% RSLogix 500 project horizontal_tank_integer.RSS, saved by version 8.30.00.16 %
PROJECT "UNTITLED"    % processor: Bul.1763 MicroLogix 1100 Series A %

PROGRAM FILES
  LAD 2   2 rungs
  LAD 255 "ONEDEPTH"  10 rungs

DATA FILES
  O0 OUTPUT  4 elements
  I1 INPUT  6 elements
  S2 STATUS  66 elements
  B3 BINARY  1 elements
  T4 TIMER  1 elements
  C5 COUNTER  1 elements
  R6 CONTROL  1 elements
  N7 INTEGER  20 elements
  F8 FLOAT  1 elements
  F254   128 elements
  N255   256 elements

LADDER 2
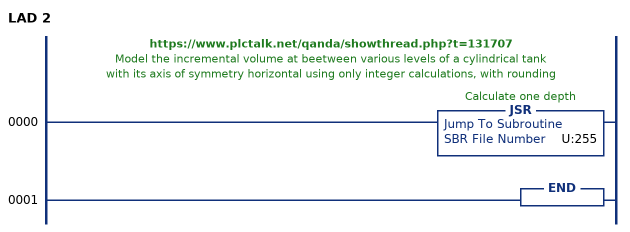
% Rung: 0 %
% TITLE: https://www.plctalk.net/qanda/showthread.php?t=131707 %
% Model the incremental volume at beetween various levels of a cylindrical tank
% with its axis of symmetry horizontal using only integer calculations, with rounding %
SOR JSR U:255 EOR
%   U:255  "Calculate one depth" %
% Rung: 1 %
SOR END EOR

LADDER 255 "ONEDEPTH"
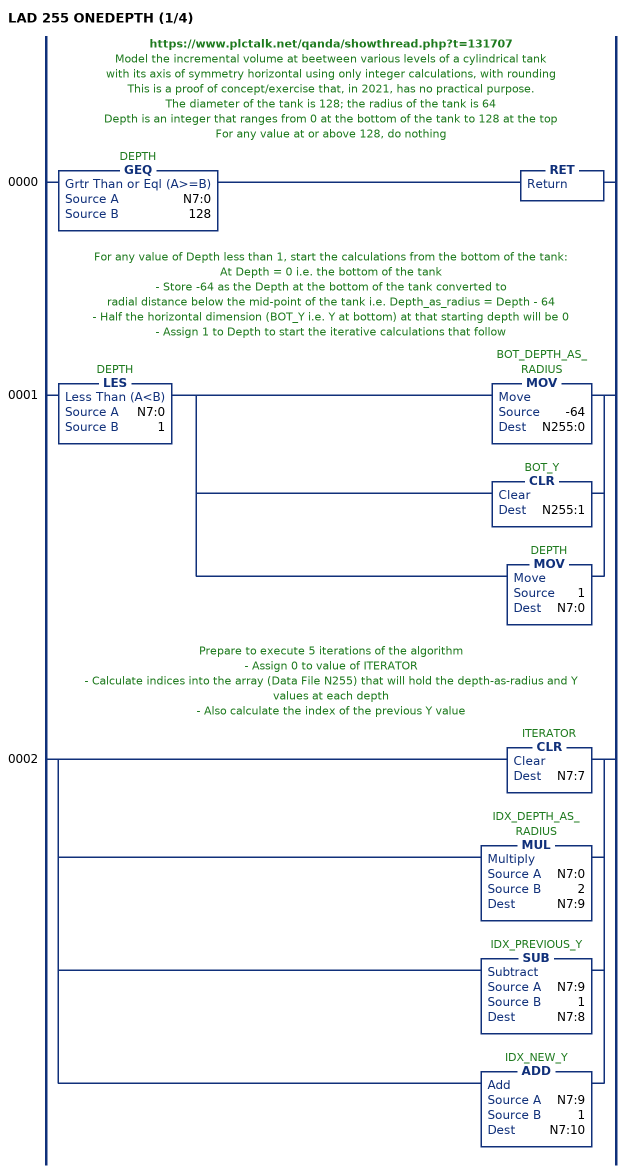
% Rung: 0 %
% TITLE: https://www.plctalk.net/qanda/showthread.php?t=131707 %
% Model the incremental volume at beetween various levels of a cylindrical tank
% with its axis of symmetry horizontal using only integer calculations, with rounding
% 
% This is a proof of concept/exercise that, in 2021, has no practical purpose.
% 
% The diameter of the tank is 128; the radius of the tank is 64
% Depth is an integer that ranges from 0 at the bottom of the tank to 128 at the top
% For any value at or above 128, do nothing %
SOR GEQ N7:0 128 RET EOR
%   N7:0  DEPTH %
% Rung: 1 %
% For any value of Depth less than 1, start the calculations from the bottom of the tank:
% At Depth = 0 i.e. the bottom of the tank
% - Store -64 as the Depth at the bottom of the tank converted to
%   radial distance below the mid-point of the tank i.e. Depth_as_radius = Depth - 64
% - Half the horizontal dimension (BOT_Y i.e. Y at bottom) at that starting depth will be 0
% - Assign 1 to Depth to start the iterative calculations that follow %
SOR LES N7:0 1 BST MOV -64 N255:0 NXB CLR N255:1 NXB MOV 1 N7:0 BND EOR
%   N7:0  DEPTH %
%   N255:0  BOT_DEPTH_AS_RADIUS %
%   N255:1  BOT_Y %
% Rung: 2 %
% Prepare to execute 5 iterations of the algorithm
% - Assign 0 to value of ITERATOR
% - Calculate indices into the array (Data File N255) that will hold the depth-as-radius and Y values at each depth
% - Also calculate the index of the previous Y value %
SOR BST CLR N7:7 NXB MUL N7:0 2 N7:9 NXB SUB N7:9 1 N7:8 NXB ADD N7:9 1 N7:10 BND EOR
%   N7:7  ITERATOR %
%   N7:0  DEPTH %
%   N7:9  IDX_DEPTH_AS_RADIUS %
%   N7:8  IDX_PREVIOUS_Y %
%   N7:10  IDX_NEW_Y %

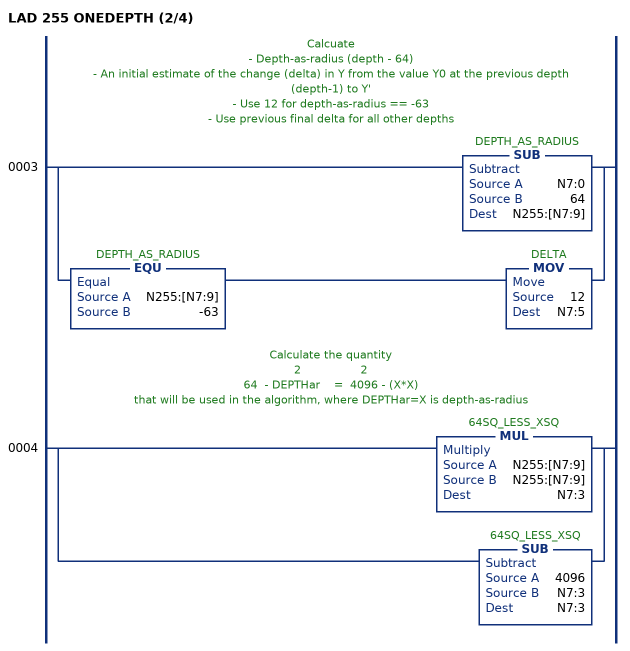
% Rung: 3 %
% Calcuate
% - Depth-as-radius (depth - 64)
% - An initial estimate of the change (delta) in Y from the value Y0 at the previous depth (depth-1) to Y'
%   - Use 12 for depth-as-radius == -63
%   - Use previous final delta for all other depths %
SOR BST SUB N7:0 64 N255:[N7:9] NXB EQU N255:[N7:9] -63 MOV 12 N7:5 BND EOR
%   N7:0  DEPTH %
%   N255:[N7:9]  DEPTH_AS_RADIUS %
%   N7:9  IDX_DEPTH_AS_RADIUS %
%   N7:5  DELTA %
% Rung: 4 %
% Calculate the quantity
% 
%      2                 2
%   64  - DEPTHar    =  4096 - (X*X)
% 
% that will be used in the algorithm, where DEPTHar=X is depth-as-radius %
SOR BST MUL N255:[N7:9] N255:[N7:9] N7:3 NXB SUB 4096 N7:3 N7:3 BND EOR
%   N255:[N7:9]  DEPTH_AS_RADIUS %
%   N7:9  IDX_DEPTH_AS_RADIUS %
%   N7:3  64SQ_LESS_XSQ %

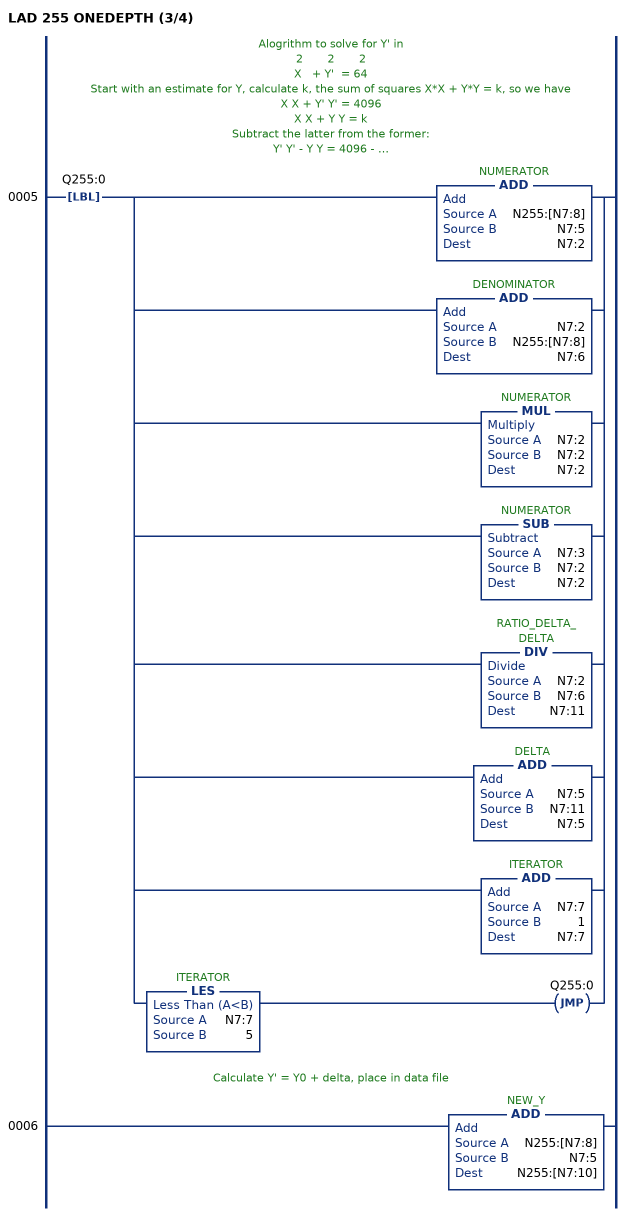
% Rung: 5 %
% Alogrithm to solve for Y' in
%       2       2       2
%     X   + Y'  = 64
% Start with an estimate for Y, calculate k, the sum of squares X*X + Y*Y = k, so we have
%    X X + Y' Y' = 4096
%    X X + Y Y = k
% Subtract the latter from the former:
%    Y' Y' - Y Y = 4096 - k
% Assume there is a difference, delta, between Y' and Y:
%   Y' = Y + delta
% Substituting
%   (Y+delta) (Y+delta) - Y Y = 4096 - k
%   Y Y + 2 Y delta + delta delta - Y*Y = 4096 - k
%   2  Y delta + delta delta = 4096 - k
%   delta (2Y + delta) = 4096 - k
%   delta = (4096 - k) / (2Y + deltaOLD)
% Use successive substitution:
% - Start with an estimate of Y as the Y0 from the previous depth,
% - Use the previous depth's delta as deltaOLD, so Y' = Y0 + deltaOLD, to calculate an incremental delta:
%   incrdelta = (4096 - k) / (2Y + deltaOLD)
% - Increment deltaOLD by incrdelta to get a new deltaOLD
%   deltaOLD = deltaOLD + incrdelta = deltaOLD + (4096 - k) / (2Y + deltaOLD)
% and repeat for five iterations %
SOR LBL Q255:0 BST ADD N255:[N7:8] N7:5 N7:2 NXB ADD N7:2 N255:[N7:8] N7:6 NXB MUL N7:2 N7:2 N7:2 NXB SUB N7:3 N7:2 N7:2 NXB DIV N7:2 N7:6 N7:11 NXB ADD N7:5 N7:11 N7:5 NXB ADD N7:7 1 N7:7 NXB LES N7:7 5 JMP Q255:0 BND EOR
%   N255:[N7:8]  PREVIOUS_Y %
%   N7:8  IDX_PREVIOUS_Y %
%   N7:5  DELTA %
%   N7:2  NUMERATOR %
%   N7:6  DENOMINATOR %
%   N7:3  64SQ_LESS_XSQ %
%   N7:11  RATIO_DELTA_DELTA %
%   N7:7  ITERATOR %
% Rung: 6 %
% Calculate Y' = Y0 + delta, place in data file %
SOR ADD N255:[N7:8] N7:5 N255:[N7:10] EOR
%   N255:[N7:8]  PREVIOUS_Y %
%   N7:8  IDX_PREVIOUS_Y %
%   N7:5  DELTA %
%   N255:[N7:10]  NEW_Y %
%   N7:10  IDX_NEW_Y %

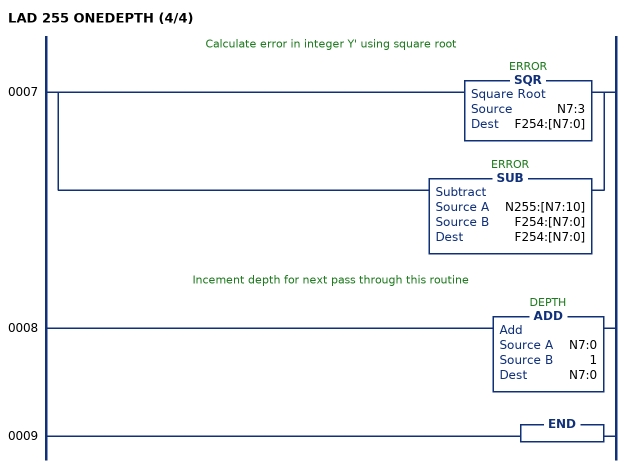
% Rung: 7 %
% Calculate error in integer Y' using square root %
SOR BST SQR N7:3 F254:[N7:0] NXB SUB N255:[N7:10] F254:[N7:0] F254:[N7:0] BND EOR
%   N7:3  64SQ_LESS_XSQ %
%   F254:[N7:0]  ERROR %
%   N7:0  DEPTH %
%   N255:[N7:10]  NEW_Y %
%   N7:10  IDX_NEW_Y %
% Rung: 8 %
% Incement depth for next pass through this routine %
SOR ADD N7:0 1 N7:0 EOR
%   N7:0  DEPTH %
% Rung: 9 %
SOR END EOR

OTHER DOCUMENTED ADDRESSES
  N7:4  RADIUS

DATA TABLE (non-zero values as saved)
DATA B3
% B3:0 % 0X0001
